PROGRAM PRG_WriteOutputs
VAR
END_VAR

GVL_IO.stOutputs.bSafetyRunRequest := GVL_MASTER.stOutputs.bSafetyRunRequest;
GVL_IO.stOutputs.bSafetyResetRequest := GVL_MASTER.stOutputs.bSafetyResetRequest;
GVL_IO.stOutputs.bSafetyErrorAcknowledgementRequest := GVL_MASTER.stOutputs.bSafetyErrorAcknowledgementRequest;
GVL_IO.stOutputs.bAirSupplyEnable := GVL_MASTER.stOutputs.bAirSupplyEnable;
GVL_IO.stOutputs.bMainDoorLockRequest := GVL_MASTER.stOutputs.bMainDoorLockRequest;
GVL_IO.stOutputs.bIndexRotatePortA := GVL_MASTER.stOutputs.bIndexRotatePortA;
GVL_IO.stOutputs.bIndexStopPortB := GVL_MASTER.stOutputs.bIndexStopPortB;

GVL_IO.stOutputs.bStation1SupportExtend := FALSE; // Removed Station 1 nest support.
GVL_IO.stOutputs.bStation1SupportRetract := FALSE; // Retired compatibility output.
GVL_IO.stOutputs.bStation2SupportExtend := GVL_MASTER.stOutputs.bStation2SupportExtend;
GVL_IO.stOutputs.bStation2SupportRetract := GVL_MASTER.stOutputs.bStation2SupportRetract;
GVL_IO.stOutputs.bStation3SupportExtend := FALSE; // Retired output.
GVL_IO.stOutputs.bStation3SupportRetract := FALSE; // Retired output.

GVL_IO.stOutputs.bVisionHorizontalBack := GVL_MASTER.stOutputs.bVisionHorizontalBack;
GVL_IO.stOutputs.bVisionHorizontalFront := GVL_MASTER.stOutputs.bVisionHorizontalFront;
GVL_IO.stOutputs.bVisionVerticalUp := GVL_MASTER.stOutputs.bVisionVerticalUp;
GVL_IO.stOutputs.bVisionVerticalDown := GVL_MASTER.stOutputs.bVisionVerticalDown;
GVL_IO.stOutputs.bVisionLimitOff := FALSE; // Retired output.
GVL_IO.stOutputs.bVisionLimitOn := FALSE; // Retired output.
GVL_IO.stOutputs.bVisionGripClose := GVL_MASTER.stOutputs.bVisionGripClose;
GVL_IO.stOutputs.bVisionGripOpen := GVL_MASTER.stOutputs.bVisionGripOpen;
GVL_IO.stOutputs.bVisionRotate0 := GVL_MASTER.stOutputs.bVisionRotate0;
GVL_IO.stOutputs.bVisionRotate180 := GVL_MASTER.stOutputs.bVisionRotate180;

GVL_IO.stOutputs.bHeatStakeHeadLock := GVL_MASTER.stOutputs.bHeatStakeHeadLock;
GVL_IO.stOutputs.bHeatStakeHeadUnlock := GVL_MASTER.stOutputs.bHeatStakeHeadUnlock;
GVL_IO.stOutputs.bHeatStakeHeadDown := GVL_MASTER.stOutputs.bHeatStakeHeadDown;
GVL_IO.stOutputs.bHeatStakeHeadUp := GVL_MASTER.stOutputs.bHeatStakeHeadUp;
GVL_IO.stOutputs.iHeatStakePressureRaw := GVL_MASTER.stOutputs.iHeatStakePressureRaw;
GVL_IO.stOutputs.bPatchDispenserAir := GVL_MASTER.stOutputs.bPatchDispenserAir;
GVL_IO.stOutputs.bPatchVerticalDown := GVL_MASTER.stOutputs.bPatchVerticalDown;
GVL_IO.stOutputs.bPatchVerticalUp := GVL_MASTER.stOutputs.bPatchVerticalUp;

GVL_IO.stOutputs.bLedStart := GVL_MASTER.stOutputs.bLedStart;
GVL_IO.stOutputs.bLedReset := GVL_MASTER.stOutputs.bLedReset;

// Patch Press has two independent physical status outputs.
GVL_IO.stOutputs.bStatusIndicatorRed := GVL_MASTER.stOutputs.bLedFail;
GVL_IO.stOutputs.bStatusIndicatorGreen := GVL_MASTER.stOutputs.bLedPass;

GVL_IO.stOutputs.bInternalLight := GVL_MASTER.stOutputs.bInternalLight;
GVL_IO.stOutputs.bNestLight := GVL_MASTER.stOutputs.bNestLight;
GVL_IO.stOutputs.uiHeatStakePwm1Raw := GVL_MASTER.stOutputs.uiHeatStakePwm1Raw;
GVL_IO.stOutputs.uiHeatStakePwm2Raw := GVL_MASTER.stOutputs.uiHeatStakePwm2Raw;

END_PROGRAM

(* stored: Version 1.1.0.1, ProductVersion 3.1.4026.18
   POU PRG_WriteOutputs: Id {44926d69-67e0-4fbe-81ef-c45a14e013c6}, SpecialFunc None *)
